// TIA Portal project "PLC_Progetto_2" (V15)

(* hardware
DEVICE "HMI_1"  KTP1000 Basic color PN
   slot 0: "HMI_1"  KTP1000 Basic color PN  6AV6 647-0AF11-3AX0  12.0.0.0
   slot 1: "HMI_RT_1"  KTP1000 Basic color PN  6AV6 647-0AF11-3AX0  12.0.0.0
   slot 5: "HMI_1.IE_CP_1"  PROFINET Interface  12.0.0.0
      slot 1: "PROFINET Interface_1"  PROFINET Interface
         slot 1: "Port_1"  Port
DEVICE "S7-1200 station_1"  S7-1200 Station
   slot 0: "Rack_0"  S7-1200 Rack  Rack  V1.0
   slot 1: "PLC_1"  CPU 1214C AC/DC/Rly  6ES7 214-1BG40-0XB0  V4.2
*)

// ===== PLC "PLC_1"  CPU 1214C AC/DC/Rly =====

VAR_GLOBAL   // PLC tag table "Default tag table"
   "1Hz_Clock" AT %M666.5 : Bool;
   "Clock_Byte" AT %MB666 : Byte;
   "Clock_10Hz" AT %M666.0 : Bool;
   "Clock_5Hz" AT %M666.1 : Bool;
   "Clock_2.5Hz" AT %M666.2 : Bool;
   "Clock_2Hz" AT %M666.3 : Bool;
   "Clock_1.25Hz" AT %M666.4 : Bool;
   "Clock_1Hz" AT %M666.5 : Bool;
   "Clock_0.625Hz" AT %M666.6 : Bool;
   "Clock_0.5Hz" AT %M666.7 : Bool;
END_VAR

DATA_BLOCK "DB"   // DB1
{ S7_Optimized_Access := 'TRUE' }
VERSION : 0.1
   VAR
      Go_Bit : Bool := false;
      Stop_Bit : Bool;
      Front_1 : Bool;
      Salto : Bool;
      Number : Int;
      Bit_1 : Bool;
      Bit_2 : Bool;
      Bit_3 : Bool;
      Bit_4 : Bool;
      Bit_5 : Bool;
      Bit_6 : Bool;
      Bit_7 : Bool;
      Bit_8 : Bool;
      Bit_9 : Bool;
      Bit_10 : Bool;
      NumVirg : Real;
      Area : Real;
      Perimetro : Real;
      Timer_Bit : Bool;
   END_VAR
BEGIN
END_DATA_BLOCK

// folder: System blocks/Program resources

DATA_BLOCK "IEC_Counter_0_DB"   // DB2
{ S7_Optimized_Access := 'TRUE' }
AUTHOR : Simatic
FAMILY : IEC
NAME : CNTR
VERSION : 1.0
// stored: InstanceOfName IEC_COUNTER
"IEC_COUNTER"
BEGIN
END_DATA_BLOCK

DATA_BLOCK "IEC_Timer_0_DB"   // DB3
{ S7_Optimized_Access := 'TRUE' }
AUTHOR : Simatic
FAMILY : IEC
NAME : IEC_TMR
VERSION : 1.0
// stored: InstanceOfName IEC_TIMER
"IEC_TIMER"
BEGIN
END_DATA_BLOCK

// folder: (top level)

ORGANIZATION_BLOCK "Main"   // OB1, LAD, ProgramCycle
TITLE = "Main Program Sweep (Cycle)"
{ S7_Optimized_Access := 'TRUE' }
VERSION : 0.1
   VAR_INPUT
      Initial_Call : Bool;   // Initial call of this OB
      Remanence : Bool;   // =True, if remanent data are available
   END_VAR
   VAR_TEMP   // added for the SCL form of the ladder/FBD networks
      _w1 : Bool;
   END_VAR
BEGIN

REGION Network 1
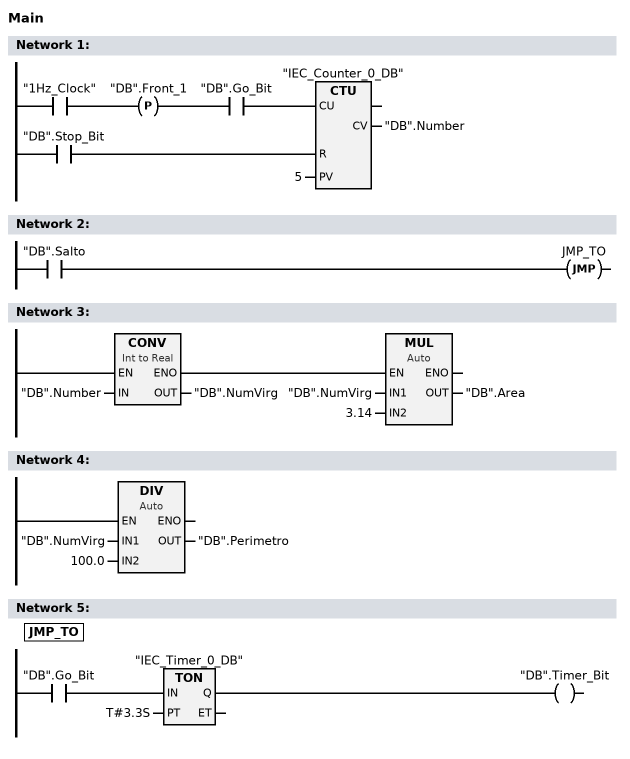
   #_w1 := "1Hz_Clock" AND NOT "DB".Front_1;   // rising edge
   "DB".Front_1 := "1Hz_Clock";
   "IEC_Counter_0_DB".CTU(CU := #_w1 AND "DB".Go_Bit, R := "DB".Stop_Bit, PV := 5, CV => "DB".Number);
END_REGION

REGION Network 2
   RUNG wire#powerrail
      Contact( "DB".Salto )
      JumpCoil( JMP_TO )
   END_RUNG
   // the same network as SCL:
   IF "DB".Salto THEN GOTO JMP_TO; END_IF;
END_REGION

REGION Network 3
   RUNG wire#powerrail
      { S7_Templates := "[SrcType := Int, DestType := Real]" } Convert(in := "DB".Number, out => "DB".NumVirg)
      Mul(in1 := "DB".NumVirg, in2 := 3.14, out => "DB".Area)
   END_RUNG
   // the same network as SCL:
   "DB".NumVirg := INT_TO_REAL("DB".Number);
   "DB".Area := "DB".NumVirg * 3.14;
END_REGION

REGION Network 4
   RUNG wire#powerrail
      Div(in1 := "DB".NumVirg, in2 := 100.0, out => "DB".Perimetro)
   END_RUNG
   // the same network as SCL:
   "DB".Perimetro := "DB".NumVirg / 100.0;
END_REGION

REGION Network 5
   JMP_TO:
   "IEC_Timer_0_DB".TON(IN := "DB".Go_Bit, PT := T#3.3S);
   "DB".Timer_Bit := "IEC_Timer_0_DB".Q;
END_REGION
END_ORGANIZATION_BLOCK

(* ===== HMI "HMI_RT_1" =====
system functions are stored by id; their names below are inferred from use
connection "HMI_Connection_1": ETHERNET, SMART_S7_1200_OMS

HMI tags "Default tag table"
   "DB_NumVirg" : Real = PLC "DB".NumVirg, 1 s
   "DB_Area" : Real = PLC "DB".Area, 1 s
   "DB_Go_Bit" : Bool = PLC "DB".Go_Bit, 1 s
   "DB_Stop_Bit" : Bool = PLC "DB".Stop_Bit, 1 s

Template "Template_1" 640x480
   Button "Exit" at 560,422 size 79x57; TextOff 'Exit'; PictureOff "ExitRuntime_KTP1000_Basic_color_PN"; PictureOn "ExitRuntime_KTP1000_Basic_color_PN"
      on Release: StopRuntime(0)
   Button "Template_Button" at 480,422 size 79x57; TextOff 'Text'
   Button "Template_Button_1" at 400,422 size 79x57; TextOff 'Text'
   Button "Template_Button_2" at 320,422 size 79x57; TextOff 'Text'
   Button "Template_Button_3" at 240,422 size 79x57; TextOff 'Text'
   Button "Template_Button_4" at 160,422 size 79x57; TextOff 'Text'
   Button "Template_Button_5" at 80,422 size 79x57; TextOff 'Text'
   Button "Start screen" at 0,422 size 79x57; TextOff 'Start screen'; PictureOff "NavigateHome_KTP1000_Basic_color_PN"; PictureOn "NavigateHome_KTP1000_Basic_color_PN"
      on Release: ActivateScreen("Root screen", 0)

screen "Root screen" 640x480, template "Template_1"
   TextField "HmiScreenItemData_1" at 59,14 size 512x22; Text 'Pagina 1'
   IOField "I/O field_1" at 373,64 size 124x40; FormatPattern 999.99
      ProcessValue <- "DB_NumVirg"
   Button "Button_1" at 22,64 size 212x37; TextOff 'START'
      on Press: InvertBit("DB_Go_Bit")
   IOField "I/O field_2" at 373,111 size 124x40; FormatPattern 999.99
      ProcessValue <- "DB_Area"
   TextField "Text field_1" at 313,76 size 60x18; Text 'NumVirg:'
   TextField "Text field_2" at 313,121 size 39x18; Text 'Area:'
   Button "Button_2" at 22,114 size 212x37; TextOff 'RESET 1/0'
      on Press: InvertBit("DB_Stop_Bit")

screen "Screen0" 640x480, template "Template_1"
   TextField "HmiScreenItemData" at 64,197 size 512x22; Text 'Screen0'
   Button "Back" at 1,1 size 159x47; TextOff 'Back'
      on Release: ActivateScreen("Root screen", 0)
*)